PROGRAM Temp_Logg
VAR
	
	fbLogg1 		:FB_SaveToCSV_Temp;
	tUpdateTime1	:TIME:=T#5S;
	sFileName1		:STRING(255):='Tempgivare';
	
	

END_VAR

fbLogg1(
	bChangeSeparatorToComma:= FALSE, 
	bExecute:= GVL_Fastighet.CSVTempProbes, 
	tUpdateTime:= tUpdateTime1, 
	sFileName:= sFileName1, 
	nDayOfWeek:= PLC_TID.fbTime.systemTime.wDayOfWeek,
	sColumn1TimeStamp:= PLC_TID.systemTime, 
	sColumn2:= REAL_TO_STRING(GVL_IO._GT41_MV), 
	sColumn3:= REAL_TO_STRING(GVL_IO._GT42_MV), 
	sColumn4:= REAL_TO_STRING(GVL_IO._GT43_MV), 
	sColumn5:= REAL_TO_STRING(GVL_IO._GT44_MV), 
	sColumn6:= REAL_TO_STRING(GVL_IO._GT45_MV), 
	sColumn7:= REAL_TO_STRING(GVL_IO._GT46_MV),
	sColumn8:= REAL_TO_STRING(GVL_IO._GT47_MV),
	sColumn9:= REAL_TO_STRING(GVL_IO._GT48_MV));

END_PROGRAM

(* stored: Version 1.1.0.1, ProductVersion 3.1.4022.3
   POU Temp_Logg: Id {1735528a-ef65-405d-8d5b-7ee34e26eb52}, SpecialFunc None *)
